FUNCTION Convert_TIME_TO_TOD : BOOL
VAR_INPUT
	in : TIME;
	out : REFERENCE TO TOD;
END_VAR
VAR
	converted : TOD;
END_VAR

converted := TIME_TO_TOD(in);

IF (TOD_TO_TIME(converted) <> in) THEN
	RETURN;
END_IF

out := converted;
Convert_TIME_TO_TOD := TRUE;

END_FUNCTION

(* stored: Version 1.1.0.1, ProductVersion 3.1.4024.12
   POU Convert_TIME_TO_TOD: Id {5e513905-b2ff-46dc-8ac0-05969a116a8f}, SpecialFunc None *)
